ABB RAPID module: Module1.mod

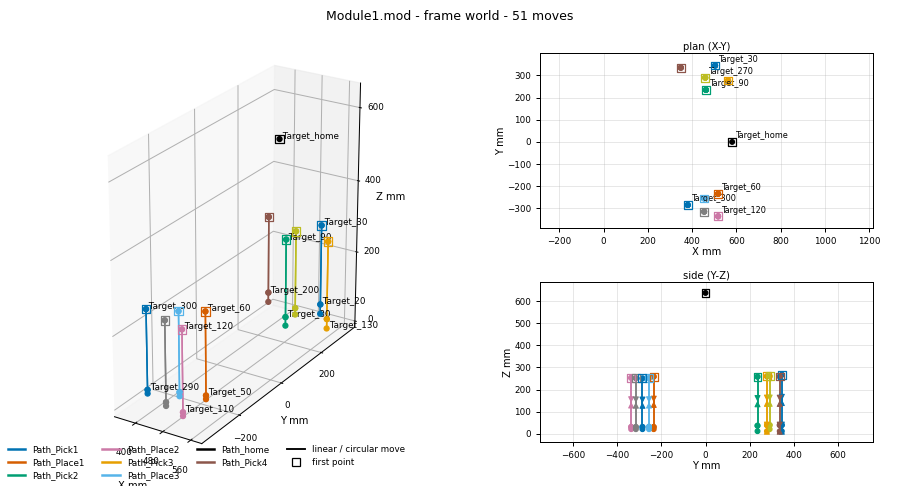
[picture p0: tool path of Module1.mod in frame world, 51 of 51 moves have a stored position in this frame; points joined in program order, loops and branches not executed]
MODULE Module1
        CONST robtarget Target_30:=[[-203.936,35,266.737020433],[0,0.949987841,0.312286892,0],[0,0,-1,0],[9E+09,9E+09,9E+09,9E+09,9E+09,9E+09]];
    CONST robtarget Target_20:=[[-203.936,35,39.153397437],[0,0.949987841,0.312286892,0],[0,0,-1,0],[9E+09,9E+09,9E+09,9E+09,9E+09,9E+09]];
    CONST robtarget Target_10:=[[-203.936,35,11.718007752],[0,0.949987841,0.312286892,0],[0,0,0,0],[9E+09,9E+09,9E+09,9E+09,9E+09,9E+09]];
    CONST robtarget Target_60:=[[-177.616,21.569,255.150981984],[0,0.945648604,0.325190279,0],[-1,0,-1,0],[9E+09,9E+09,9E+09,9E+09,9E+09,9E+09]];
    CONST robtarget Target_50:=[[-177.616,21.569,27.931115203],[0,0.945648604,0.325190279,0],[-1,0,-1,0],[9E+09,9E+09,9E+09,9E+09,9E+09,9E+09]];
    CONST robtarget Target_40:=[[-177.616,21.569,17.782272012],[0,0.945648604,0.325190279,0],[0,0,0,0],[9E+09,9E+09,9E+09,9E+09,9E+09,9E+09]];
    CONST robtarget Target_90:=[[-162.526,145,258.022987661],[0,0.969025845,0.246959333,0],[0,0,-1,0],[9E+09,9E+09,9E+09,9E+09,9E+09,9E+09]];
    CONST robtarget Target_80:=[[-162.526,145,36.604094028],[0,0.969025845,0.246959333,0],[0,0,-1,0],[9E+09,9E+09,9E+09,9E+09,9E+09,9E+09]];
    CONST robtarget Target_70:=[[-162.526,145,11.718007752],[0,0.969025845,0.246959333,0],[0,0,0,0],[9E+09,9E+09,9E+09,9E+09,9E+09,9E+09]];
    CONST robtarget Target_120:=[[-177.616,123.605,249.729565319],[0,0.972297946,0.233744957,0],[-1,0,-1,0],[9E+09,9E+09,9E+09,9E+09,9E+09,9E+09]];
    CONST robtarget Target_110:=[[-177.616,123.605,28.106578616],[0,0.972297946,0.233744957,0],[-1,0,-1,0],[9E+09,9E+09,9E+09,9E+09,9E+09,9E+09]];
    CONST robtarget Target_100:=[[-177.616,123.605,17.782272012],[0,0.972297946,0.233744957,0],[0,0,0,0],[9E+09,9E+09,9E+09,9E+09,9E+09,9E+09]];
    CONST robtarget Target_150:=[[-262.397,102.45,259.896311518],[0,0.949987841,0.312286892,0],[0,0,-1,0],[9E+09,9E+09,9E+09,9E+09,9E+09,9E+09]];
    CONST robtarget Target_140:=[[-262.397,102.45,38.974527513],[0,0.949987841,0.312286892,0],[0,0,-1,0],[9E+09,9E+09,9E+09,9E+09,9E+09,9E+09]];
    CONST robtarget Target_130:=[[-262.397,102.45,11.718007752],[0,0.949987841,0.312286892,0],[0,0,0,0],[9E+09,9E+09,9E+09,9E+09,9E+09,9E+09]];
    CONST robtarget Target_180:=[[-114.445,42.918,248.469873973],[0,-0.240856605,0.970560712,0],[-1,0,1,0],[9E+09,9E+09,9E+09,9E+09,9E+09,9E+09]];
    CONST robtarget Target_170:=[[-114.445,42.918,29.074547572],[0,-0.240856605,0.970560712,0],[-1,0,1,0],[9E+09,9E+09,9E+09,9E+09,9E+09,9E+09]];
    CONST robtarget Target_160:=[[-114.445,42.918,17.682272012],[0,-0.240856605,0.970560712,0],[0,0,0,0],[9E+09,9E+09,9E+09,9E+09,9E+09,9E+09]];
    CONST robtarget Target_home:=[[580.769835971,0,636.5],[0.5,0,0.866025404,0],[0,0,0,0],[9E+09,9E+09,9E+09,9E+09,9E+09,9E+09]];
    CONST robtarget Target_210:=[[-49.151,44.642,258.937140242],[0,0.949987841,0.312286892,0],[0,0,0,0],[9E+09,9E+09,9E+09,9E+09,9E+09,9E+09]];
    CONST robtarget Target_200:=[[-49.151,44.642,39.041514377],[0,0.949987841,0.312286892,0],[0,0,0,0],[9E+09,9E+09,9E+09,9E+09,9E+09,9E+09]];
    CONST robtarget Target_190:=[[-49.151,44.642,11.618007752],[0,0.949987841,0.312286892,0],[0,0,0,0],[9E+09,9E+09,9E+09,9E+09,9E+09,9E+09]];
    CONST robtarget Target_240:=[[-114.445,102.256,248.45188105],[0,0.736771325,-0.676142008,0],[0,0,0,0],[9E+09,9E+09,9E+09,9E+09,9E+09,9E+09]];
    CONST robtarget Target_230:=[[-114.445,102.256,27.852777925],[0,0.736771325,-0.676142008,0],[-1,0,0,0],[9E+09,9E+09,9E+09,9E+09,9E+09,9E+09]];
    CONST robtarget Target_220:=[[-114.445,102.256,17.682272012],[0,0.736771325,-0.676142008,0],[-1,0,0,0],[9E+09,9E+09,9E+09,9E+09,9E+09,9E+09]];
    CONST robtarget Target_270:=[[-159.395,90,260.079399122],[0,0.949987841,0.312286892,0],[0,0,0,0],[9E+09,9E+09,9E+09,9E+09,9E+09,9E+09]];
    CONST robtarget Target_260:=[[-159.395,90,39.22173393],[0,0.949987841,0.312286892,0],[0,0,-1,0],[9E+09,9E+09,9E+09,9E+09,9E+09,9E+09]];
    CONST robtarget Target_250:=[[-159.395,90,20.618007752],[0,0.949987841,0.312286892,0],[0,0,-1,0],[9E+09,9E+09,9E+09,9E+09,9E+09,9E+09]];
    CONST robtarget Target_300:=[[-40.25,72.587,247.204652011],[0,0.949987841,0.312286892,0],[0,0,0,0],[9E+09,9E+09,9E+09,9E+09,9E+09,9E+09]];
    CONST robtarget Target_290:=[[-40.25,72.587,27.948178752],[0,0.949987841,0.312286892,0],[-1,0,-1,0],[9E+09,9E+09,9E+09,9E+09,9E+09,9E+09]];
    CONST robtarget Target_280:=[[-40.25,72.587,17.682272012],[0,0.949987841,0.312286892,0],[-1,0,-1,0],[9E+09,9E+09,9E+09,9E+09,9E+09,9E+09]];
!***********************************************************
    !
    ! Module:  Module1
    !
    ! Description:
    !   <Insert description here>
    !
    ! Author: danny
    !
    ! Version: 1.0
    !
    !***********************************************************


    !***********************************************************
    !
    ! Procedure main
    !
    !   This is the entry point of your program
    !
    !***********************************************************
    PROC main()
        WaitDI DI_01,1;
        Ensamble1;
    ENDPROC
    PROC Ensamble1()
        Path_home;
        Path_Pick2;
        Path_Place2;
        Path_Pick1;
        Path_Place1;
        Path_Pick3;
        Path_Place3;
        Path_Pick4;
        Path_Place4;
        Path_Pick5;
        Path_Place5;
        Path_home;
    ENDPROC

    PROC Path_Pick1()
        MoveL Target_30,v200,z0,T_ventosa\WObj:=WO_Peak;
        MoveL Target_20,v200,z0,T_ventosa\WObj:=WO_Peak;
        MoveL Target_10,v200,z0,T_ventosa\WObj:=WO_Peak;
        SetDO DO_02,0;
        SetDO DO_01,1;
        WaitTime 1;
        MoveL Target_20,v200,z0,T_ventosa\WObj:=WO_Peak;
        MoveL Target_30,v200,z0,T_ventosa\WObj:=WO_Peak;
    ENDPROC
    PROC Path_Place1()
        MoveL Target_60,v200,z0,T_ventosa\WObj:=WO_Place;
        MoveL Target_50,v200,z0,T_ventosa\WObj:=WO_Place;
        MoveL Target_40,v200,z0,T_ventosa\WObj:=WO_Place;
        SetDO DO_01,0;
        SetDO DO_02,1;
        WaitTime 1;
        MoveL Target_50,v200,z0,T_ventosa\WObj:=WO_Place;
        MoveL Target_60,v200,z0,T_ventosa\WObj:=WO_Place;
    ENDPROC
    PROC Path_Pick2()
        MoveL Target_90,v200,z0,T_ventosa\WObj:=WO_Peak;
        MoveL Target_80,v200,z0,T_ventosa\WObj:=WO_Peak;
        MoveL Target_70,v200,z0,T_ventosa\WObj:=WO_Peak;
        SetDO DO_02,0;
        SetDO DO_01,1;
        WaitTime 1;
        MoveL Target_80,v200,z0,T_ventosa\WObj:=WO_Peak;
        MoveL Target_90,v200,z0,T_ventosa\WObj:=WO_Peak;
    ENDPROC
    PROC Path_Place2()
        MoveL Target_120,v200,z0,T_ventosa\WObj:=WO_Place;
        MoveL Target_110,v200,z0,T_ventosa\WObj:=WO_Place;
        MoveL Target_100,v200,z0,T_ventosa\WObj:=WO_Place;
        SetDO DO_01,0;
        SetDO DO_02,1;
        WaitTime 1;
        MoveL Target_110,v200,z0,T_ventosa\WObj:=WO_Place;
        MoveL Target_120,v200,z0,T_ventosa\WObj:=WO_Place;
    ENDPROC
    PROC Path_Pick3()
        MoveL Target_150,v200,z0,T_ventosa\WObj:=WO_Peak;
        MoveL Target_140,v200,z0,T_ventosa\WObj:=WO_Peak;
        MoveL Target_130,v200,z0,T_ventosa\WObj:=WO_Peak;
        SetDO DO_02,0;
        SetDO DO_01,1;
        WaitTime 1;
        MoveL Target_140,v200,z0,T_ventosa\WObj:=WO_Peak;
        MoveL Target_150,v200,z0,T_ventosa\WObj:=WO_Peak;
    ENDPROC
    PROC Path_Place3()
        MoveJ Target_180,v200,z0,T_ventosa\WObj:=WO_Place;
        MoveL Target_170,v200,z0,T_ventosa\WObj:=WO_Place;
        MoveL Target_160,v200,z0,T_ventosa\WObj:=WO_Place;
        SetDO DO_01,0;
        SetDO DO_02,1;
        WaitTime 1;
        MoveL Target_170,v200,z0,T_ventosa\WObj:=WO_Place;
        MoveL Target_180,v200,z0,T_ventosa\WObj:=WO_Place;
    ENDPROC
    PROC Path_home()
        MoveJ Target_home,v200,z0,T_ventosa\WObj:=wobj0;
    ENDPROC
    PROC Path_Pick4()
        MoveJ Target_210,v200,z0,T_ventosa\WObj:=WO_Peak;
        MoveL Target_200,v200,z0,T_ventosa\WObj:=WO_Peak;
        MoveL Target_190,v200,z0,T_ventosa\WObj:=WO_Peak;
        SetDO DO_02,0;
        SetDO DO_01,1;
        WaitTime 1;
        MoveL Target_200,v200,z0,T_ventosa\WObj:=WO_Peak;
        MoveL Target_210,v200,z0,T_ventosa\WObj:=WO_Peak;
    ENDPROC
    PROC Path_Place4()
        MoveJ Target_240,v200,z0,T_ventosa\WObj:=WO_Place;
        MoveL Target_230,v200,z0,T_ventosa\WObj:=WO_Place;
        MoveL Target_220,v200,z0,T_ventosa\WObj:=WO_Place;
        SetDO DO_01,0;
        SetDO DO_02,1;
        WaitTime 1;
        MoveL Target_230,v200,z0,T_ventosa\WObj:=WO_Place;
        MoveL Target_240,v200,z0,T_ventosa\WObj:=WO_Place;
    ENDPROC
    PROC Path_Pick5()
        MoveJ Target_270,v200,z0,T_ventosa\WObj:=WO_Peak;
        MoveL Target_260,v200,z0,T_ventosa\WObj:=WO_Peak;
        MoveL Target_250,v200,z0,T_ventosa\WObj:=WO_Peak;
        SetDO DO_02,0;
        SetDO DO_01,1;
        WaitTime 1;
        MoveL Target_260,v200,z0,T_ventosa\WObj:=WO_Peak;
        MoveL Target_270,v200,z0,T_ventosa\WObj:=WO_Peak;
    ENDPROC
    PROC Path_Place5()
        MoveL Target_300,v200,z0,T_ventosa\WObj:=WO_Place;
        MoveL Target_290,v200,z0,T_ventosa\WObj:=WO_Place;
        MoveL Target_280,v200,z0,T_ventosa\WObj:=WO_Place;
        SetDO DO_01,0;
        SetDO DO_02,1;
        WaitTime 1;
        MoveL Target_290,v200,z0,T_ventosa\WObj:=WO_Place;
        MoveL Target_300,v200,z0,T_ventosa\WObj:=WO_Place;
    ENDPROC
ENDMODULE
